Omron CX-Programmer project NewProject (CX-Programmer 9.75)

# PLC NewPLC1: CP1L M

## Global symbols (name address type ; comment)
0.00 BOOL  ; Sensor-1
0.01 BOOL  ; Sensor-2
0.02 BOOL  ; Sensor-3
0.03 BOOL  ; LS-1
0.04 BOOL  ; LS-2
100.00 BOOL  ; Open
100.01 BOOL  ; Close
W0.00 BOOL  ; In / Out

## Program NewProgram1 (cyclic task 0)

### Section Section1

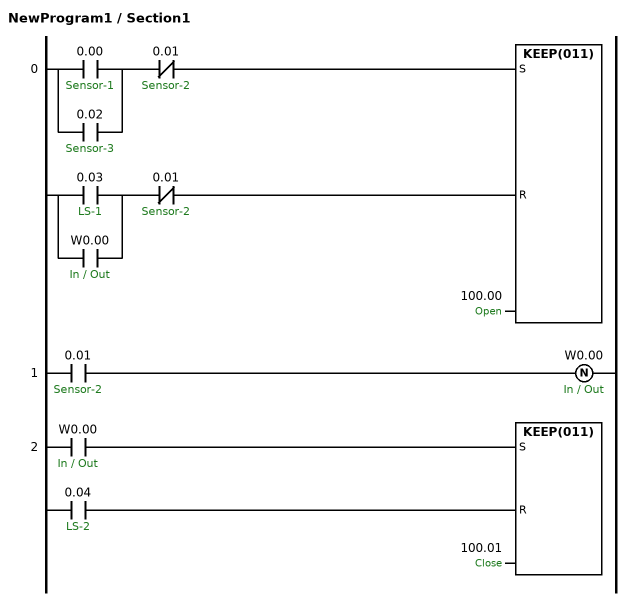
; rung 0
LD 0.00  ; Sensor-1
OR 0.02  ; Sensor-3
ANDNOT 0.01  ; Sensor-2
LD 0.03  ; LS-1
OR W0.00  ; In / Out
ANDNOT 0.01  ; Sensor-2
KEEP(011) 100.00  ; Open
; rung 1
LD 0.01  ; Sensor-2
DIFD(014) W0.00  ; In / Out
; rung 2
LD W0.00  ; In / Out
LD 0.04  ; LS-2
KEEP(011) 100.01  ; Close

### Section END
; rung 0
END(001)